(* PLC project electric_jack, Dassault Systèmes ControlBuild 2024x *)
(* stored: creationDateTime 2023-10-03T11:13:07-01:00 *)

(* This module simulates an electric jack and its electrical logic control *)
FUNCTION_BLOCK equipment_library.electric_jack
  VAR_INPUT
    voltage380 : BOOL := true;
    cmdSupply : BOOL := true;
    sensorSupply : BOOL := true;
  END_VAR
  VAR_INPUT
    valveWork : BOOL := false;
    valveRest : BOOL := false;
  END_VAR
  VAR_OUTPUT
    outletSensor : BOOL := false;
    inletSensor : BOOL := false;
    valveOpen : BOOL := false;
    valveClosed : BOOL := false;
    thermal : BOOL := false;
  END_VAR
  VAR_OUTPUT
    rodPosition : REAL := 0.0;
    rodPercent : REAL := 0.0;
    incrementValue : REAL := 0.0;
  END_VAR
  VAR
    closeState : BOOL := false;
    openState : BOOL := false;
    increment : REAL := 0.0;
    memoClose : BOOL := false;
    memoOpen : BOOL := false;
  END_VAR
  VAR CONSTANT
    inletSensorLogic : BOOL := true;
    outletSensorLogic : BOOL := true;
    openLogic : BOOL := true;
    closeLogic : BOOL := true;
    thermalLogic : BOOL := false;
    rodLength : REAL := 1000.0;
    time2extend : REAL := 2.0;
  END_VAR
  VAR
    d_electrical : BOOL := false;
    v_d_electrical : BOOL := true;
    d_valveClose : BOOL := false;
    v_d_valveClose : BOOL := false;
    d_valveOpen : BOOL := false;
    v_d_valveOpen : BOOL := false;
    d_outletSensor : BOOL := false;
    v_d_outletSensor : BOOL := false;
    d_inletSensor : BOOL := false;
    v_d_inletSensor : BOOL := false;
    d_locking : BOOL := false;
    v_d_locking : REAL := 0.0;
  END_VAR


ACTION C_source_code:
/* ----------------------------------------------------------------	*/
/* Type : Model of Operative Behaviour					*/
/* Category :  Associations - Jacks					*/
/* Author : Dassault Systemes						*/
/* Update date : June 2018							*/
/* ----------------------------------------------------------------	*/
/* This module simulates an electric jack and its electrical 		*/
/* logic control.								*/
/* ----------------------------------------------------------------	*/

/* ----------------------------------------------------------------	*/
/* Management of orders from Control Part					*/
/*	if there is no power supply for command the solenoid 		*/
/*     control valve doesn't understand the control order.		*/
/* ----------------------------------------------------------------	*/
if (valveWork && !memoClose && cmdSupply) memoOpen = 1;
if (!valveWork || !cmdSupply) memoOpen = 0;
if (!memoOpen && valveRest && cmdSupply) memoClose = 1;
if (!valveRest || !cmdSupply) memoClose = 0;

/* ----------------------------------------------------------------	*/
/* Calculation of the on-state of contactors				*/
/* ----------------------------------------------------------------	*/
openState = memoOpen & voltage380 & ! d_electrical;
closeState = memoClose & voltage380 & ! d_electrical;

/* ----------------------------------------------------------------	*/
/* Management of the rod evolution						*/
/* the rod stays in its current position if there is no pressure 	*/
/* in the two chambers. 							*/
/* ----------------------------------------------------------------	*/
incrementValue = 0;
if (! d_locking)  {
	if (time2extend > 0.0)
		increment = (rodLength/time2extend)*(CLOCK_PERIOD/1000000);
	if (openState && ! closeState ) {
		if ( rodPosition < rodLength ) {
			(rodPosition) += increment;
			incrementValue = increment;
		}
		if ( rodPosition > rodLength ) {
			incrementValue -= rodPosition - rodLength;
			rodPosition = rodLength;
		}
	}
	if (closeState && ! openState ) {
		if ( rodPosition > 0 ) {
			(rodPosition) -= increment;
			incrementValue = increment * -1.0;
		}
		if ( rodPosition < 0.0 ) {
			incrementValue -= rodPosition;
			rodPosition = 0.0;
		}
	}
}

/* ----------------------------------------------------------------	*/
/* Calculation of the rod position in percentage			*/
/* ----------------------------------------------------------------	*/
if (rodLength != 0.0)
	rodPercent = ((rodPosition/rodLength)*100);

/* ----------------------------------------------------------------	*/
/* Management of the thermal sensor					*/
/* ----------------------------------------------------------------	*/
if (d_electrical) thermal = v_d_electrical;
else
	thermal = ! thermalLogic && sensorSupply;

/* ----------------------------------------------------------------	*/
/* Management of the contactors feed-backs				*/
/* ----------------------------------------------------------------	*/
if (d_valveOpen) valveOpen = v_d_valveOpen;
else
	valveOpen = (memoOpen ^ ! openLogic) && sensorSupply;

if (d_valveClose) valveClosed = v_d_valveClose;
else
	valveClosed = (memoClose ^ ! closeLogic) && sensorSupply;

/* ----------------------------------------------------------------	*/
/* Management of the sensors state						*/
/* ----------------------------------------------------------------	*/
if (d_outletSensor) outletSensor = v_d_outletSensor;
else
	outletSensor = ((rodPosition >= rodLength) ^ ! outletSensorLogic) && sensorSupply;

if (d_inletSensor) inletSensor = v_d_inletSensor;
else
	inletSensor = ((rodPosition <= 0) ^ ! inletSensorLogic) && sensorSupply;
END_ACTION
END_FUNCTION_BLOCK
